TYPE ST_Euchner_MGB2_HW_IN :
STRUCT
	///Hardware In
	nByte0: USINT;
	///Hardware In
	nByte1: USINT;
END_STRUCT
END_TYPE

(* stored: Version 1.1.0.1, ProductVersion 3.1.4024.12
   DUT ST_Euchner_MGB2_HW_IN: Id {2216d48b-7684-4a74-a5af-768362594d1a} *)
